// TIA Portal V17 export
// export: Created 2021-12-03T08:13:03.4298677Z, ExportSetting WithDefaults, DisplayName Totally Integrated Automation Portal, DisplayVersion V17, DisplayName TIA Portal Openness, DisplayVersion V17, DisplayName TIA Portal Version Control Interface, DisplayVersion V17, DisplayName STEP 7 Professional, DisplayVersion V17, DisplayName STEP 7 Safety, DisplayVersion V17, DisplayName WinCC Advanced, DisplayVersion V17
DATA_BLOCK "DBI_MN_Acc_Ctrl"   // DB62
VERSION : 0.1
// stored: AutoNumber false, InstanceOfName FB_MN_Acc_Ctrl, InstanceOfType FB
"FB_MN_Acc_Ctrl"
   // VAR_INPUT
   //    I_InitTrue { ExternalVisible := 'False'; ExternalWritable := 'False'} : Bool;
   //    I_Acc_PwrOnRq { ExternalVisible := 'False'; ExternalWritable := 'False'} : Bool;
   //    I_AccChil_PwrIsOn { ExternalVisible := 'False'; ExternalWritable := 'False'} : Bool;
   //    I_Mod220V_PwrIsOn { ExternalVisible := 'False'; ExternalWritable := 'False'} : Bool;
   //    I_Mod380V_PwrIsOn { ExternalVisible := 'False'; ExternalWritable := 'False'} : Bool;
   //    I_AccCS_PrwIsOn { ExternalVisible := 'False'; ExternalWritable := 'False'} : Bool;
   //    I_AccRemMode { ExternalVisible := 'False'; ExternalWritable := 'False'} : Bool;
   //    I_AccWarmUp { ExternalVisible := 'False'; ExternalWritable := 'False'} : Bool;
   //    I_AccClear { ExternalVisible := 'False'; ExternalWritable := 'False'} : Bool;
   //    I_AccStandby { ExternalVisible := 'False'; ExternalWritable := 'False'} : Bool;
   //    I_AccReady { ExternalVisible := 'False'; ExternalWritable := 'False'} : Bool;
   //    I_RFOn_Rq { ExternalVisible := 'False'; ExternalWritable := 'False'} : Bool;
   //    I_XRay_Rq { ExternalVisible := 'False'; ExternalWritable := 'False'} : Bool;
   //    I_Acc_PwrOffRq { ExternalVisible := 'False'; ExternalWritable := 'False'} : Bool;
   //    I_ChillOffDly { ExternalVisible := 'False'; ExternalWritable := 'False'} : Bool;
   //    I_AccFault { ExternalVisible := 'False'; ExternalWritable := 'False'} : Bool;
   //    I_NOEStop { ExternalVisible := 'False'; ExternalWritable := 'False'} : Bool;
   //    I_FltRst { ExternalVisible := 'False'; ExternalWritable := 'False'} : Bool;
   //    I_FullWarmUp { ExternalVisible := 'False'; ExternalWritable := 'False'} : Bool;
   //    I_SafePeriIsCls { ExternalVisible := 'False'; ExternalWritable := 'False'} : Bool;
   //    I_PwrRst { ExternalVisible := 'False'; ExternalWritable := 'False'} : Bool;
   // END_VAR
   // VAR_OUTPUT
   //    O_AccPreh_PwrOn { ExternalVisible := 'False'; ExternalWritable := 'False'} : Bool;
   //    O_Mod380V_RlyOn { ExternalVisible := 'False'; ExternalWritable := 'False'} : Bool;
   //    O_AccMod220V_PwrOn { ExternalVisible := 'False'; ExternalWritable := 'False'} : Bool;
   //    O_Chil_PwrOn { ExternalVisible := 'False'; ExternalWritable := 'False'} : Bool;
   //    O_FltRst { ExternalVisible := 'False'; ExternalWritable := 'False'} : Bool;
   //    O_WarmUp { ExternalVisible := 'False'; ExternalWritable := 'False'} : Bool;
   //    O_RFOn { ExternalVisible := 'False'; ExternalWritable := 'False'} : Bool;
   //    O_XRay_On { ExternalVisible := 'False'; ExternalWritable := 'False'} : Bool;
   //    O_FullWarmUp_Rq { ExternalVisible := 'False'; ExternalWritable := 'False'} : Bool;
   //    O_Acc_ActState { ExternalVisible := 'False'; ExternalWritable := 'False'} : Int;
   // END_VAR
   // VAR RETAIN
   //    S_PwrRst { ExternalVisible := 'False'} : Bool;
   //    AxSR { ExternalVisible := 'False'; ExternalWritable := 'False'} : Struct
   //       Acc230V_PwrOn { ExternalVisible := 'False'; ExternalWritable := 'False'} : Bool;
   //    END_STRUCT;
   //    S_Transit { ExternalVisible := 'False'; ExternalWritable := 'False'} : Struct
   //       InitTrue { ExternalVisible := 'False'; ExternalWritable := 'False'} : Bool;
   //       ReqAccPwrOn { ExternalVisible := 'False'; ExternalWritable := 'False'} : Bool;
   //       ChillOnDly { ExternalVisible := 'False'; ExternalWritable := 'False'} : Bool;
   //       ModOnDly { ExternalVisible := 'False'; ExternalWritable := 'False'} : Bool;
   //       AccPrwOn { ExternalVisible := 'False'; ExternalWritable := 'False'} : Bool;
   //       NAccPrwOn { ExternalVisible := 'False'; ExternalWritable := 'False'} : Bool;
   //       AccRemMode { ExternalVisible := 'False'; ExternalWritable := 'False'} : Bool;
   //       NAccRemMode { ExternalVisible := 'False'; ExternalWritable := 'False'} : Bool;
   //       AccWarmUp { ExternalVisible := 'False'; ExternalWritable := 'False'} : Bool;
   //       AccClear { ExternalVisible := 'False'; ExternalWritable := 'False'} : Bool;
   //       AccStandby { ExternalVisible := 'False'; ExternalWritable := 'False'} : Bool;
   //       AccReady { ExternalVisible := 'False'; ExternalWritable := 'False'} : Bool;
   //       AccRfOn { ExternalVisible := 'False'; ExternalWritable := 'False'} : Bool;
   //       AccRfOff { ExternalVisible := 'False'; ExternalWritable := 'False'} : Bool;
   //       AccXrayOn { ExternalVisible := 'False'; ExternalWritable := 'False'} : Bool;
   //       AccXrayOff { ExternalVisible := 'False'; ExternalWritable := 'False'} : Bool;
   //       ReqAccPwrOff { ExternalVisible := 'False'; ExternalWritable := 'False'} : Bool;
   //       AccNotActive { ExternalVisible := 'False'; ExternalWritable := 'False'} : Bool;
   //       XrayHeadOffDly { ExternalVisible := 'False'; ExternalWritable := 'False'} : Bool;
   //       ModOffDly { ExternalVisible := 'False'; ExternalWritable := 'False'} : Bool;
   //       ChillOffDly { ExternalVisible := 'False'; ExternalWritable := 'False'} : Bool;
   //       AccFault { ExternalVisible := 'False'; ExternalWritable := 'False'} : Bool;
   //       ACK_AccFault { ExternalVisible := 'False'; ExternalWritable := 'False'} : Bool;
   //       EStop { ExternalVisible := 'False'; ExternalWritable := 'False'} : Bool;
   //    END_STRUCT;
   //    DI_Acc_StateCase { ExternalVisible := 'False'; S7_SetPoint := 'True'} : "FB_Acc_StateCase";
   //    S_Acc_ActState { ExternalVisible := 'False'; ExternalWritable := 'False'} : Int;
   // END_VAR
BEGIN
END_DATA_BLOCK
